// TwinCAT 3 PLC project PLC1
// ProgramVersion: 3.1.4023.0
// libraries:
//   Tc2_Standard, * (Beckhoff Automation GmbH)
//   Tc2_System, * (Beckhoff Automation GmbH)
//   Tc2_Utilities, * (Beckhoff Automation GmbH)
//   Tc3_IotBase, * (Beckhoff Automation GmbH)
//   Tc3_JsonXml, * (Beckhoff Automation GmbH)
//   Tc3_Module, * (Beckhoff Automation GmbH)
// project tree:
//   / PlcTask.TcTTO
//   POUs/ FB_HttpGet.TcPOU, FB_HttpPut.TcPOU, MAIN.TcPOU
// real-time tasks:
//   TASK PlcTask: cycle T#100us, priority 20, ADS port 350

CONFIGURATION PLC1
    RESOURCE PLC ON TwinCAT3
        TASK PlcTask(INTERVAL := T#100us, PRIORITY := 20);
        PROGRAM MAIN WITH PlcTask : MAIN;
    END_RESOURCE
END_CONFIGURATION

// ---- POUs/MAIN.TcPOU
PROGRAM MAIN
VAR
	fbHttpClient: FB_IotHttpClient := (sHostName:= '192.168.1.99',bKeepAlive := TRUE, tConnectionTimeout:=T#10S);
	bExecute: BOOL := TRUE;

	fbPut: FB_HttpPut;
	fbGet: FB_HttpGet;
	bPut: BOOL;
	bGet: BOOL;
	
	bwOn: BOOL := TRUE; 
	nwSat: USINT := 254;
	nwBri: USINT := 140;
    nwHue: UINT := 1;
	nwTrans: UINT := 1;
	swEffect: STRING[10] := 'none';
	
	brOn: BOOL ;
	nrSat: USINT ;
	nrBri: USINT;
    nrHue: UINT;
	nrTrans: UINT;
	srEffect: STRING[10] ;
	
	fbTimer: ton := (pt:=T#100MS);
END_VAR

IF NOT fbHttpClient.bConfigured THEN
	fbHttpClient.nHostPort := 80;
	fbHttpClient.stTLS.bNoServerCertCheck:= TRUE;
END_IF

IF fbHttpClient.bConfigured THEN
	fbPut(bSend:= bPut, bOn:= bwOn, nSat:= nwSat, nBri:= nwBri, nHue:= nwHue, nTrans:= nwTrans, sEffect:= swEffect,fbClient:= fbHttpClient);
	fbGet(bGet := bGet, bOn=> brOn, nSat=> nrSat, nBri=> nrBri, nHue=> nrHue, sEffect=> srEffect,fbClient:= fbHttpClient);
END_IF

IF bExecute THEN
	IF bPut THEN
		bPut:= FALSE;
		bExecute:= FALSE;
	END_IF
	IF bGet THEN
		bGet := FALSE;
		bExecute:= FALSE;
		nrTrans := nwTrans;
	END_IF
END_IF

fbHttpClient.Execute();

END_PROGRAM

// ---- POUs/FB_HttpPut.TcPOU
FUNCTION_BLOCK FB_HttpPut
VAR_INPUT
	bSend: BOOL;
	bOn: BOOL; 
	nSat: USINT;
	nBri: USINT;
    nHue: UINT;
	nTrans: UINT;
	sEffect: STRING[10];
		
END_VAR
VAR_IN_OUT
	fbClient             : FB_IotHttpClient;
END_VAR
VAR_OUTPUT
	bBusy                : BOOL;
    bError               : BOOL;
END_VAR
VAR
	fbRequest: FB_IotHttpRequest;
	//fbJson: FB_JsonDomParser;
	fbJsonWriter: FB_JsonSaxWriter;
	nState: UDINT;
	RisingEdge: R_TRIG;
	
	sContent: STRING(511);
	sSend: STRING(511);
	
	//jsonDoc: SJsonValue;
	//jsonVal: SJsonValue;
	//sResultValue: STRING;

END_VAR

RisingEdge(clk:= bSend);

CASE nState OF
0: 
	fbJsonWriter.StartObject();
	fbJsonWriter.AddKey('on');
	fbJsonWriter.AddBool(bOn);	
	fbJsonWriter.AddKey('sat');
	fbJsonWriter.AddUdint(nSat);
	fbJsonWriter.AddKey('bri');
	fbJsonWriter.AddUdint(nBri);
	fbJsonWriter.AddKey('hue');
	fbJsonWriter.AddUdint(nHue);
	fbJsonWriter.AddKey('transitiontime');
	fbJsonWriter.AddUdint(nTrans);
	fbJsonWriter.AddKey('effect');
	fbJsonWriter.AddString(sEffect);
	fbJsonWriter.EndObject();
	sSend:= fbJsonWriter.GetDocument();
	fbJsonWriter.ResetDocument();
	
	IF RisingEdge.Q THEN
		IF fbRequest.SendRequest(sUri:='/api/OOrb8w4GpeITNRtK0w5Yf6Ke3p1k6PnnwycVn68a/lights/4/state', 
			fbClient:=fbClient, eRequestType:= ETcIotHttpRequestType.HTTP_PUT,
			pContent:= ADR(sSend), nContentSize:= LEN2(ADR(sSend)), 0) THEN
			
			nState:= 1;
			bBusy:= TRUE;
			bError:= FALSE;
		END_IF
	END_IF
	
1:
	IF NOT fbRequest.bBusy THEN
		bError:= TRUE;
		IF NOT fbRequest.bError THEN
			fbRequest.GetContent(pContent:= ADR(sContent), nContentSize:= SIZEOF(sContent), bSetNullTermination:= TRUE);
			IF fbRequest.nStatusCode >= 200 AND fbRequest.nStatusCode < 300 THEN              
                bError:= FALSE;    
            END_IF
        END_IF
        nState:= 0;
        bBusy:= FALSE;
	END_IF
END_CASE

END_FUNCTION_BLOCK

// ---- POUs/FB_HttpGet.TcPOU
FUNCTION_BLOCK FB_HttpGet
VAR_INPUT
	bGet: BOOL;
END_VAR
VAR_IN_OUT	
	fbClient             : FB_IotHttpClient;
END_VAR
VAR_OUTPUT
	bBusy                : BOOL;
    bError               : BOOL;
	
	bOn: BOOL; 
	nSat: USINT;
	nBri: USINT;
    nHue: UINT;
	sEffect: STRING[10];
END_VAR
VAR
	fbRequest: FB_IotHttpRequest;
	fbJson: FB_JsonDomParser;
	fbJsonWriter: FB_JsonSaxWriter;
	nState: UDINT;
	RisingEdge: R_TRIG;
	
	sContent: STRING(511);
	sSend: STRING(511);
	
	jsonDoc: SJsonValue;
	jsonState: SJsonValue;
	jsonOn: SJsonValue;
	jsonSat: SJsonValue;
	jsonBri: SJsonValue;
	jsonHue: SJsonValue;
	jsonEffect: SJsonValue;
END_VAR

RisingEdge(CLK:= bGet);

CASE nState OF
0:
    IF RisingEdge.Q THEN
        IF fbRequest.SendRequest(sUri:= '/api/OOrb8w4GpeITNRtK0w5Yf6Ke3p1k6PnnwycVn68a/lights/4',
            fbClient:= fbClient, eRequestType:= ETcIotHttpRequestType.HTTP_Get, 
			0, 0, 0) THEN
			
            nState:= 1;
            bBusy:= TRUE;
            bError:= FALSE;
        END_IF
    END_IF
1:
    IF NOT fbRequest.bBusy THEN
        bError:= TRUE;
        IF NOT fbRequest.bError THEN
            fbRequest.GetContent(pContent:= ADR(sContent), nContentSize:= SIZEOF(sContent), bSetNullTermination:= TRUE);
            IF fbRequest.nStatusCode >= 200 AND fbRequest.nStatusCode < 300 THEN
                jsonDoc:= fbRequest.GetJsonDomContent(fbJson);
                IF jsonDoc <> 0 THEN
					
					IF fbJson.HasMember(jsonDoc,'state') THEN
						jsonState:= fbJson.FindMember(jsonDoc, 'state');
						IF fbJson.HasMember(jsonState, 'on') THEN
							jsonOn:= fbJson.FindMember(jsonState, 'on');
							IF fbJson.IsBool(jsonOn) THEN
								bOn:= fbJson.GetBool(jsonOn);
							END_IF
						END_IF	
						IF fbJson.HasMember(jsonState, 'sat') THEN
							jsonSat:= fbJson.FindMember(jsonState, 'sat');
							IF fbJson.IsUint(jsonSat) THEN
								nSat:= UDINT_TO_USINT(fbJson.GetUint(jsonSat));
							END_IF
						END_IF	
						IF fbJson.HasMember(jsonState, 'bri') THEN
							jsonBri:= fbJson.FindMember(jsonState, 'bri');
							IF fbJson.IsUint(jsonBri) THEN
								nBri:= UDINT_TO_USINT(fbJson.GetUint(jsonBri));
							END_IF
						END_IF	
						IF fbJson.HasMember(jsonState, 'hue') THEN
							jsonHue:= fbJson.FindMember(jsonState, 'hue');
							IF fbJson.IsUint(jsonHue) THEN
								nHue:= UDINT_TO_UINT(fbJson.GetUint(jsonHue));
							END_IF
						END_IF	
						IF fbJson.HasMember(jsonState, 'effect') THEN
							jsonEffect:= fbJson.FindMember(jsonState, 'effect');
							IF fbJson.IsString(jsonEffect) THEN
								sEffect:= fbJson.Getstring(jsonEffect);
							END_IF
						END_IF	
						
						bError:= FALSE;					
					END_IF
                END_IF
            END_IF
        END_IF
        nState:= 0;
        bBusy:= FALSE;
    END_IF
END_CASE

END_FUNCTION_BLOCK
